VAR_GLOBAL CONSTANT
    // 设备最大轴数量。
    cMaxAxisCount : UINT := 14;
END_VAR

(* stored: Version 1.1.0.1, ProductVersion 3.1.4026.18
   GVL GVL_Constants: Id {79aafccb-e265-458e-9299-9ce99396c7cf} *)
